# EPICS StreamDevice protocol: siteApps/cryomodule-1-0/proto/temperature.proto
terminator = CR LF;

replytimeout = 3000;
readtimeout = 1000;

read_kelvin {out "KRDG? \$1"; in "%f";}
reset {out "*RST";}
self_test {out "TST?"; in "%f";}
get_comm {out "LEDS?"; in "%f";}
